// TIA Portal V20 export
DATA_BLOCK "ControlNodes"   // DB171
// stored: MemoryReserve 100, Namespace Unit1.Em2
   VAR
      em { ExternalWritable := 'False'} : "LAF_typeEmControlNode";
      cm { ExternalWritable := 'False'} : "Unit1.Em2.typeCmControlNode";
      citiMap : "LER_OEM_Data";
      SemiAutuSplice { ExternalWritable := 'False'} : "Unit1.Em2.typeSequenceControlNode";
   END_VAR
   VAR RETAIN
      cmElectrodeFixRightTopFwdBwd { ExternalWritable := 'False'} : "LBC_typeTwoWayActuatorControlNode";
      cmElectrodeFixRightBottomFwdBwd { ExternalWritable := 'False'} : "LBC_typeTwoWayActuatorControlNode";
      cmElectrodeFixLeftTopFwdBwd { ExternalWritable := 'False'} : "LBC_typeTwoWayActuatorControlNode";
      cmElectrodeFixLeftBottomFwdBwd { ExternalWritable := 'False'} : "LBC_typeTwoWayActuatorControlNode";
      cmElectrodeFixLeftTopUpDown { ExternalWritable := 'False'} : "LBC_typeTwoWayActuatorControlNode";
      cmElectrodeFixLeftBottomUpDown { ExternalWritable := 'False'} : "LBC_typeTwoWayActuatorControlNode";
      cmUwSemiSplicerVacuumRightTopOnOff { ExternalWritable := 'False'} : "LBC_typeTwoWayActuatorControlNode";
      cmUwSemiSplicerVacuumRightBottomOnOff { ExternalWritable := 'False'} : "LBC_typeTwoWayActuatorControlNode";
      cmUwSemiSplicerVacuumLeftTopOnOff { ExternalWritable := 'False'} : "LBC_typeTwoWayActuatorControlNode";
      cmUwSemiSplicerVacuumLeftBottomOnOff { ExternalWritable := 'False'} : "LBC_typeTwoWayActuatorControlNode";
      cmElectrodeCutterFwdBwd { ExternalWritable := 'False'} : "LBC_typeTwoWayActuatorControlNode";
      cmSplicingLeftModuleMoverFwdBwd { ExternalWritable := 'False'} : "LBC_typeTwoWayActuatorControlNode";
      cmSplicingRightModuleMoverFwdBwd { ExternalWritable := 'False'} : "LBC_typeTwoWayActuatorControlNode";
      cmElectrodeLeftHolderMoverFwdBwd { ExternalWritable := 'False'} : "LBC_typeTwoWayActuatorControlNode";
      cmElectrodeRightHolderMoverFwdBwd { ExternalWritable := 'False'} : "LBC_typeTwoWayActuatorControlNode";
      cmTapeLoadingTurnCwCcw { ExternalWritable := 'False'} : "LBC_typeTwoWayActuatorControlNode";
      cmTapeAttachUnitFwdBwd { ExternalWritable := 'False'} : "LBC_typeTwoWayActuatorControlNode";
      cmTapeVacuumOnOff { ExternalWritable := 'False'} : "LBC_typeTwoWayActuatorControlNode";
      cmStopperFwdBwd { ExternalWritable := 'False'} : "LBC_typeTwoWayActuatorControlNode";
      cmSupportUnitTransferFwdBwd { ExternalWritable := 'False'} : "LBC_typeTwoWayActuatorControlNode";
      cmSupportUnitShaftUpDown { ExternalWritable := 'False'} : "LBC_typeTwoWayActuatorControlNode";
      cmFrameCoverFwdBwd { ExternalWritable := 'False'} : "LBC_typeTwoWayActuatorControlNode";
   END_VAR
   VAR
      TapeAttachRetryCountPV { ExternalWritable := 'False'} : Int;
   END_VAR
BEGIN
END_DATA_BLOCK
